// TIA Portal V16 export
// export: Created 2021-07-12T14:47:16.7130255Z, ExportSetting WithDefaults, DisplayName Totally Integrated Automation Portal, DisplayVersion V16, DisplayName TIA Portal Version Control Interface, DisplayVersion V16, DisplayName TIA Portal Openness, DisplayVersion V16, DisplayName STEP 7 Professional, DisplayVersion V16, DisplayName STEP 7 Safety, DisplayVersion V16, DisplayName WinCC Professional, DisplayVersion V16
DATA_BLOCK "SimaHydTO_AxisBasics_PosAxis_DB"   // DB2
FAMILY : SimaHydTO/LAxisBasics
VERSION : 1.0
// stored: AutoNumber true, DBAccessibleFromOPCUA true, InstanceOfName SimaHydTO_AxisBasics_PosAxis, InstanceOfType FB
"SimaHydTO_AxisBasics_PosAxis"
   // VAR_INPUT
   //    axis : TO_PositioningAxis;
   //    powerEnable : Bool;
   //    powerStartMode : DInt;
   //    powerStopMode : Int;
   //    resetExecute : Bool;
   //    resetRestart : Bool;
   //    homeExecute : Bool;
   //    homePosition : LReal;
   //    homeMode : Int;
   //    jogForward : Bool;
   //    jogBackward : Bool;
   //    jogVelocity : LReal;
   //    jogAcceleration : LReal;
   //    jogDeceleration : LReal;
   //    jogJerk : LReal;
   //    jogPositionControlled : Bool;
   // END_VAR
   // VAR_OUTPUT
   //    powerStatus { ExternalWritable := 'False'} : Bool;
   //    powerBusy { ExternalWritable := 'False'} : Bool;
   //    resetDone { ExternalWritable := 'False'} : Bool;
   //    resetBusy { ExternalWritable := 'False'} : Bool;
   //    homeDone { ExternalWritable := 'False'} : Bool;
   //    homeBusy { ExternalWritable := 'False'} : Bool;
   //    jogInVelocity { ExternalWritable := 'False'} : Bool;
   //    jogBusy { ExternalWritable := 'False'} : Bool;
   //    commandAborted { ExternalWritable := 'False'} : Bool;
   //    error { ExternalWritable := 'False'} : Bool;
   //    errorID { ExternalWritable := 'False'} : Word;
   //    statusID { ExternalWritable := 'False'} : Int;
   // END_VAR
   // VAR
   //    instMcPower { ExternalAccessible := 'False'; ExternalVisible := 'False'; ExternalWritable := 'False'; S7_SetPoint := 'True'} : MC_POWER;
   //    instMcReset { ExternalAccessible := 'False'; ExternalVisible := 'False'; ExternalWritable := 'False'; S7_SetPoint := 'True'} : MC_RESET;
   //    instMcHome { ExternalAccessible := 'False'; ExternalVisible := 'False'; ExternalWritable := 'False'; S7_SetPoint := 'True'} : MC_HOME;
   //    instMcMoveJog { ExternalAccessible := 'False'; ExternalVisible := 'False'; ExternalWritable := 'False'; S7_SetPoint := 'True'} : MC_MOVEJOG;
   //    statCommandAborted { ExternalAccessible := 'False'; ExternalVisible := 'False'; ExternalWritable := 'False'} : Array[1..32] of Bool;
   //    statError { ExternalAccessible := 'False'; ExternalVisible := 'False'; ExternalWritable := 'False'} : Array[1..32] of Bool;
   //    statErrorID { ExternalAccessible := 'False'; ExternalVisible := 'False'; ExternalWritable := 'False'} : Array[1..32] of Word;
   //    MC_MOVEABSOLUTE_Instance { S7_SetPoint := 'True'} : MC_MOVEABSOLUTE;
   // END_VAR
BEGIN
END_DATA_BLOCK
